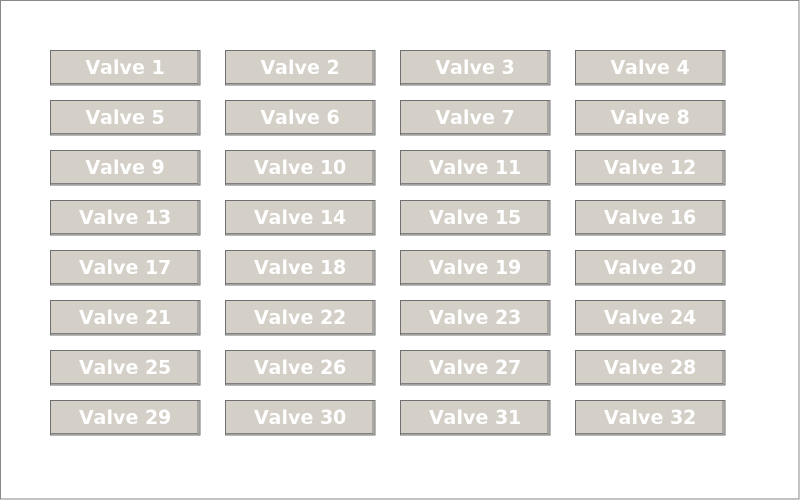
VISUALIZATION Screen_1_Sub_1  // 800x500
    Button (50,50 150x35), "Valve 1", colour toggle: GVL.HMI_Button_Valve[0]
        toggle GVL.HMI_Button_Valve[0] p2164770859=TRUE
    Button (225,50 150x35), "Valve 2", colour toggle: GVL.HMI_Button_Valve[1]
        toggle GVL.HMI_Button_Valve[1] p2164770859=TRUE
    Button (400,50 150x35), "Valve 3", colour toggle: GVL.HMI_Button_Valve[2]
        toggle GVL.HMI_Button_Valve[2] p2164770859=TRUE
    Button (575,50 150x35), "Valve 4", colour toggle: GVL.HMI_Button_Valve[3]
        toggle GVL.HMI_Button_Valve[3] p2164770859=TRUE
    Button (50,100 150x35), "Valve 5", colour toggle: GVL.HMI_Button_Valve[4]
        toggle GVL.HMI_Button_Valve[4] p2164770859=TRUE
    Button (225,100 150x35), "Valve 6", colour toggle: GVL.HMI_Button_Valve[5]
        toggle GVL.HMI_Button_Valve[5] p2164770859=TRUE
    Button (400,100 150x35), "Valve 7", colour toggle: GVL.HMI_Button_Valve[6]
        toggle GVL.HMI_Button_Valve[6] p2164770859=TRUE
    Button (575,100 150x35), "Valve 8", colour toggle: GVL.HMI_Button_Valve[7]
        toggle GVL.HMI_Button_Valve[7] p2164770859=TRUE
    Button (50,150 150x35), "Valve 9", colour toggle: GVL.HMI_Button_Valve[8]
        toggle GVL.HMI_Button_Valve[8] p2164770859=TRUE
    Button (225,150 150x35), "Valve 10", colour toggle: GVL.HMI_Button_Valve[9]
        toggle GVL.HMI_Button_Valve[9] p2164770859=TRUE
    Button (400,150 150x35), "Valve 11", colour toggle: GVL.HMI_Button_Valve[10]
        toggle GVL.HMI_Button_Valve[10] p2164770859=TRUE
    Button (575,150 150x35), "Valve 12", colour toggle: GVL.HMI_Button_Valve[11]
        toggle GVL.HMI_Button_Valve[11] p2164770859=TRUE
    Button (50,200 150x35), "Valve 13", colour toggle: GVL.HMI_Button_Valve[12]
        toggle GVL.HMI_Button_Valve[12] p2164770859=TRUE
    Button (225,200 150x35), "Valve 14", colour toggle: GVL.HMI_Button_Valve[13]
        toggle GVL.HMI_Button_Valve[13] p2164770859=TRUE
    Button (400,200 150x35), "Valve 15", colour toggle: GVL.HMI_Button_Valve[14]
        toggle GVL.HMI_Button_Valve[14] p2164770859=TRUE
    Button (575,200 150x35), "Valve 16", colour toggle: GVL.HMI_Button_Valve[15]
        toggle GVL.HMI_Button_Valve[15] p2164770859=TRUE
    Button (50,250 150x35), "Valve 17", colour toggle: GVL.HMI_Button_Valve[16]
        toggle GVL.HMI_Button_Valve[16] p2164770859=TRUE
    Button (225,250 150x35), "Valve 18", colour toggle: GVL.HMI_Button_Valve[17]
        toggle GVL.HMI_Button_Valve[17] p2164770859=TRUE
    Button (400,250 150x35), "Valve 19", colour toggle: GVL.HMI_Button_Valve[18]
        toggle GVL.HMI_Button_Valve[18] p2164770859=TRUE
    Button (575,250 150x35), "Valve 20", colour toggle: GVL.HMI_Button_Valve[19]
        toggle GVL.HMI_Button_Valve[19] p2164770859=TRUE
    Button (50,300 150x35), "Valve 21", colour toggle: GVL.HMI_Button_Valve[20]
        toggle GVL.HMI_Button_Valve[20] p2164770859=TRUE
    Button (225,300 150x35), "Valve 22", colour toggle: GVL.HMI_Button_Valve[21]
        toggle GVL.HMI_Button_Valve[21] p2164770859=TRUE
    Button (400,300 150x35), "Valve 23", colour toggle: GVL.HMI_Button_Valve[22]
        toggle GVL.HMI_Button_Valve[22] p2164770859=TRUE
    Button (575,300 150x35), "Valve 24", colour toggle: GVL.HMI_Button_Valve[23]
        toggle GVL.HMI_Button_Valve[23] p2164770859=TRUE
    Button (50,350 150x35), "Valve 25", colour toggle: GVL.HMI_Button_Valve[24]
        toggle GVL.HMI_Button_Valve[24] p2164770859=TRUE
    Button (225,350 150x35), "Valve 26", colour toggle: GVL.HMI_Button_Valve[25]
        toggle GVL.HMI_Button_Valve[25] p2164770859=TRUE
    Button (400,350 150x35), "Valve 27", colour toggle: GVL.HMI_Button_Valve[26]
        toggle GVL.HMI_Button_Valve[26] p2164770859=TRUE
    Button (575,350 150x35), "Valve 28", colour toggle: GVL.HMI_Button_Valve[27]
        toggle GVL.HMI_Button_Valve[27] p2164770859=TRUE
    Button (50,400 150x35), "Valve 29", colour toggle: GVL.HMI_Button_Valve[28]
        toggle GVL.HMI_Button_Valve[28] p2164770859=TRUE
    Button (225,400 150x35), "Valve 30", colour toggle: GVL.HMI_Button_Valve[29]
        toggle GVL.HMI_Button_Valve[29] p2164770859=TRUE
    Button (400,400 150x35), "Valve 31", colour toggle: GVL.HMI_Button_Valve[30]
        toggle GVL.HMI_Button_Valve[30] p2164770859=TRUE
    Button (575,400 150x35), "Valve 32", colour toggle: GVL.HMI_Button_Valve[31]
        toggle GVL.HMI_Button_Valve[31] p2164770859=TRUE
END_VISUALIZATION

(* stored: Version 1.1.0.1, ProductVersion 3.1.4024.12
   Visu Screen_1_Sub_1: Id {be1127d5-979c-485f-96a6-75858626f613} *)
